// TIA Portal V20 export
// export: Created 2026-07-14T14:39:13.0692745Z, ExportSetting WithDefaults, DisplayName Totally Integrated Automation Portal, DisplayVersion V20 Update 5, DisplayName TIA Portal Openness, DisplayVersion V20 Update 4, DisplayName TIA Portal Version Control Interface, DisplayVersion V20 Update 5, DisplayName SINAMICS Startdrive Advanced, DisplayVersion V20, DisplayName SINAMICS DCC, DisplayVersion V20, DisplayName SINAMICS Startdrive G130, G150, S120, S150, SINAMICS MV, G220, S200, S210, DisplayVersion V20, DisplayName SINAMICS Startdrive G110M, G120, G120C, G120D, G120P, G115D, DisplayVersion V20, DisplayName STEP 7 Professional, DisplayVersion V20 Update 5, DisplayName STEP 7 Safety, DisplayVersion V20 Update 2, DisplayName WinCC Basic/Comfort/Advanced, DisplayVersion V20 Update 5, DisplayName WinCC Unified, DisplayVersion V20 Update 5
FUNCTION "TimingAndCalls" : Void   // FC24, LAD
{ S7_Optimized_Access := 'TRUE' }
VERSION : 0.1
// Timer/block-call reference examples (TONR/TOF/CALL)
// stored: AutoNumber true, IsIECCheckEnabled false, SetENOAutomatically false, UDAEnableTagReadback false
   VAR_TEMP
      RunEnable : Bool;
      ResetRequest : Bool;
      RunTimePreset : Time;
      HoldEnable : Bool;
      HoldTimePreset : Time;
      RawValue : Real;
      ScaleMax : Real;
      ScaledValue : Real;
   END_VAR
BEGIN

REGION Network 1: Run time accumulation (TONR)
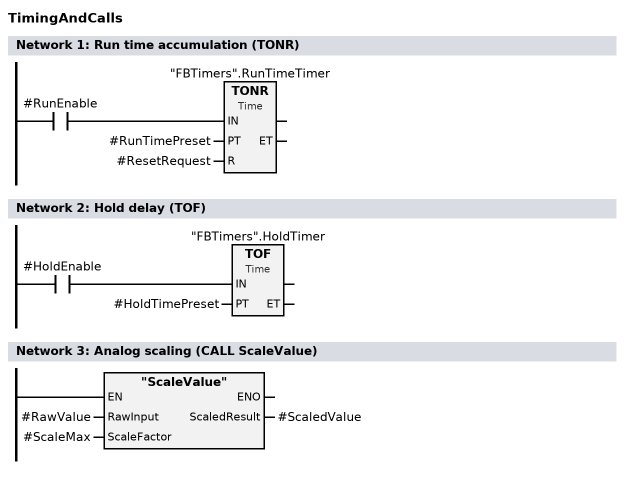
   RUNG wire#powerrail
      Contact( #RunEnable )
      { S7_Templates := "time_type := Time" } "FBTimers".RunTimeTimer.TONR(pt := #RunTimePreset, et =>, r := #ResetRequest)
   END_RUNG
   // the same network as SCL:
   "FBTimers".RunTimeTimer.TONR(IN := #RunEnable, PT := #RunTimePreset, R := #ResetRequest);
END_REGION

REGION Network 2: Hold delay (TOF)
   RUNG wire#powerrail
      Contact( #HoldEnable )
      { S7_Templates := "time_type := Time" } "FBTimers".HoldTimer.TOF(pt := #HoldTimePreset, et =>)
   END_RUNG
   // the same network as SCL:
   "FBTimers".HoldTimer.TOF(IN := #HoldEnable, PT := #HoldTimePreset);
END_REGION

REGION Network 3: Analog scaling (CALL ScaleValue)
   RUNG wire#powerrail
      "ScaleValue"(RawInput := #RawValue, ScaleFactor := #ScaleMax, ScaledResult => #ScaledValue)
   END_RUNG
   // the same network as SCL:
   "ScaleValue"(RawInput := #RawValue, ScaleFactor := #ScaleMax, ScaledResult => #ScaledValue);
END_REGION
END_FUNCTION
